{attribute 'strict'}
{attribute 'to_string'}
TYPE E_ADS_Cmd :
(
	NoCmd,
	Read,
	Write
);
END_TYPE

(* stored: Version 1.1.0.1, ProductVersion 3.1.4024.10
   EnumerationTextList E_ADS_Cmd: Id {c373949b-ed94-44f5-a1f7-a8544aaf3163} *)
